// TIA Portal V18 export
DATA_BLOCK "FB5-Dearing with valveA_DB"   // DB4
VERSION : 0.1
// stored: AutoNumber true, DBAccessibleFromOPCUA true, InstanceOfName FB5-Dearing with valve, InstanceOfType FB
"FB5-Dearing with valve"
   // VAR_INPUT
   //    "Time" : DInt;
   //    "Pump ON delay" : DInt;
   //    "Pump OFF delay" : DInt;
   // END_VAR
   // VAR_OUTPUT
   //    "dispensing Time PV" : Int;
   // END_VAR
   // VAR_IN_OUT
   //    "Start Dearing" : Bool;
   //    "Stop Dearing" : Bool;
   //    "Dearing Running" : Bool;
   //    "Dearing completed" : Bool;
   //    "ON Gear Pump" : Bool;
   //    "ON valve" : Bool;
   // END_VAR
   // VAR
   //    "dispensing time done" : Bool;
   //    "dispensing time in sec" : DInt;
   //    "timer in sec" : DInt;
   //    "timer PV in sec" : DInt;
   //    "timer input" : DInt;
   //    IEC_Timer_0_Instance { S7_SetPoint := 'True'} : TON_TIME;
   //    IEC_Timer_0_Instance_1 { S7_SetPoint := 'True'} : TON_TIME;
   //    IEC_Timer_0_Instance_2 { S7_SetPoint := 'True'} : TON_TIME;
   //    IEC_Timer_0_Instance_3 { S7_SetPoint := 'True'} : TON_TIME;
   // END_VAR
BEGIN
END_DATA_BLOCK
